TYPE DeltaMotionParameters_typ :
STRUCT
	
	Jerk			: LREAL;					// mm/s3
	Acceleration	: LREAL;					// mm/s2
	Deceleration	: LREAL;					// mm/s2
	Velocity		: LREAL;					// mm/s
	BlendingRadius	: LREAL;					// mm

END_STRUCT
END_TYPE

(* stored: Version 1.1.0.1, ProductVersion 3.1.4024.11
   DUT DeltaMotionParameters_typ: Id {424aadfa-8287-4470-a607-14095ccdc485} *)
